{attribute 'GeneratedUsingTerminal: EPP3744-0041-0016'}
{attribute addProperty BoxType "EPP3744-0041-0016"}
{attribute addProperty Id "OutputAT %Q*ARRAY[0..1] OF BOOL2"}
{attribute addProperty CRC "2036329114"}
{attribute addProperty Size "2"}
TYPE DIG_Outputs_DE230DD5 :
STRUCT
	{attribute addProperty Name "Output"}
	Output AT %Q* : ARRAY[0..1] OF BOOL;
END_STRUCT
END_TYPE

(* stored: Version 1.2.0.0, ProductVersion 3.1.4024.9
   DUT DIG_Outputs_DE230DD5: Id {b2020ce5-0420-4590-839a-b4b4991b93c6} *)
